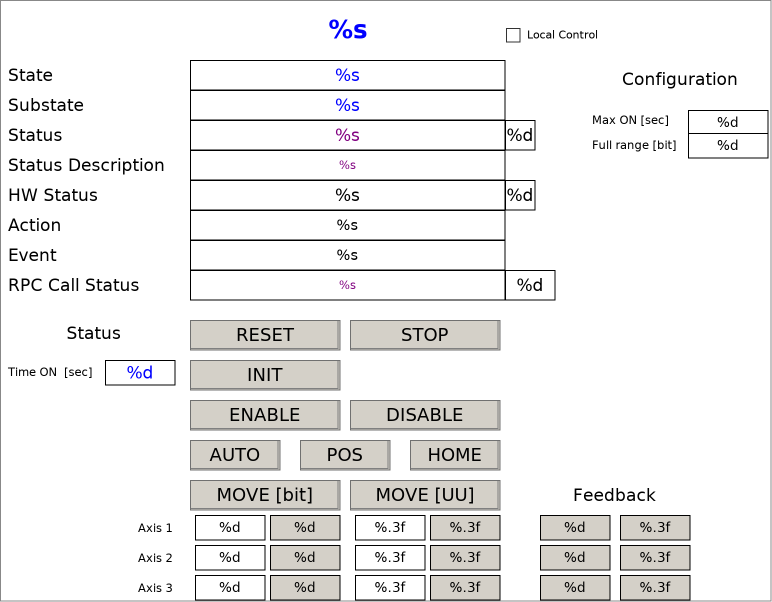
VISUALIZATION GUI_TEMPLATE_PIEZO  // 772x602
VAR_IN_OUT
	m_Instance:	FB_PIEZO_BASE;
END_VAR
    Rectangle (190,60 315x30), "%s", text variable: m_Instance.stat.sState
    Rectangle (190,90 315x30), "%s", text variable: m_Instance.stat.sSubstate
    Button (190,320 150x30), "RESET", input disabled if: (m_Instance.stat.bLocal = FALSE) <> 0
        OnMouseDown: execute { m_Instance.ctrl.nCommand := E_PIEZO_COMMAND.RESET; m_Instance.ctrl.bExecute := TRUE; }
    Button (190,360 150x30), "INIT", input disabled if: (m_Instance.stat.bLocal = FALSE) <> 0
        OnMouseDown: execute { m_Instance.ctrl.nCommand := E_PIEZO_COMMAND.INIT; m_Instance.ctrl.bExecute := TRUE; }
    Button (350,320 150x30), "STOP", input disabled if: (m_Instance.stat.bLocal = FALSE) <> 0
        OnMouseDown: execute { m_Instance.ctrl.nCommand := E_PIEZO_COMMAND.STOP; m_Instance.ctrl.bExecute := TRUE; }
    Button (190,400 150x30), "ENABLE", input disabled if: (m_Instance.stat.bLocal = FALSE) <> 0
        OnMouseDown: execute { m_Instance.ctrl.nCommand := E_PIEZO_COMMAND.ENABLE; m_Instance.ctrl.bExecute := TRUE; }
    Button (350,400 150x30), "DISABLE", input disabled if: (m_Instance.stat.bLocal = FALSE) <> 0
        OnMouseDown: execute { m_Instance.ctrl.nCommand := E_PIEZO_COMMAND.DISABLE; m_Instance.ctrl.bExecute := TRUE; }
    Button (190,440 90x30), "AUTO", tooltip "Start AUTO mode", input disabled if: (m_Instance.stat.bLocal = FALSE) <> 0
        OnMouseDown: execute { m_Instance.ctrl.nCommand := E_PIEZO_COMMAND.AUTO; m_Instance.ctrl.bExecute := TRUE; }
    Button (300,440 90x30), "POS", tooltip "Stop AUTO mode, if running. Keep piezos where they are.", input disabled if: (m_Instance.stat.bLocal = FALSE) <> 0
        OnMouseDown: execute { m_Instance.ctrl.nCommand := E_PIEZO_COMMAND.POS; m_Instance.ctrl.bExecute := TRUE; }
    Rectangle (5,60 180x30), "State"
    Rectangle (5,90 180x30), "Substate"
    Rectangle (190,120 315x30), "%s", text variable: m_Instance.stat.sStatus
    Rectangle (190,150 315x30), "%s", text variable: m_Instance.stat.sErrorText
    Rectangle (5,120 180x30), "Status"
    Rectangle (5,150 180x30), "Status Description"
    Rectangle (190,210 315x30), "%s", text variable: m_Instance.stat.sActionDesc
    Rectangle (190,240 315x30), "%s", text variable: m_Instance.stat.sEventDesc
    Rectangle (190,180 315x30), "%s", text variable: m_Instance.stat.sHwStatus
    Rectangle (5,180 180x30), "HW Status"
    Rectangle (505,180 30x30), "%d", tooltip "HW Status Index", text variable: m_Instance.stat.nHwStatus
    Rectangle (5,210 180x30), "Action"
    Rectangle (5,240 180x30), "Event"
    Rectangle (232,12 232x35), "%s", text variable: m_Instance.cfg.sName
    Rectangle (590,64 180x30), "Configuration"
    Rectangle (589,110 155x20), "Max ON [sec]"
    Rectangle (589,135 155x20), "Full range [bit]"
    Rectangle (688,110 80x25), "%d", tooltip "Maximum allowed time for lamp to be ON [sec] (>=0). Zero means no limit.", text variable: m_Instance.cfg.nMaxOn, input disabled if: (m_Instance.stat.bLocal = FALSE) <> 0
        OnMouseDown: write the text variable via Default, min 0
    Rectangle (688,133 80x25), "%d", tooltip "Full range of A/D converter controlling the intensity [bit]. Examples: 12 bit A/D = 4095 15 bit A/D = 32767 16 bit A/D = 65535", text variable: m_Instance.cfg.nFullRange[0].nValue, input disabled if: (m_Instance.stat.bLocal = FALSE) <> 0
        OnMouseDown: write the text variable via Default, min 0
    Checkbox (504,20 116x30), "Local Control", variable: m_Instance.stat.bLocal
    Rectangle (48,318 92x30), "Status"
    Rectangle (105,360 70x25), "%d", tooltip "Time since last ON command [sec]. Updated only if MaxON > 0.", text variable: m_Instance.stat.nTimeOn
    Rectangle (5,357 95x30), "Time ON [sec]"
    Rectangle (505,120 30x30), "%d", text variable: m_Instance.stat.nStatus
    Button (190,480 150x30), "MOVE [bit]", input disabled if: (m_Instance.stat.bLocal = FALSE) <> 0
        OnMouseDown: execute { m_Instance.ctrl.nCommand := E_PIEZO_COMMAND.MOVE_BIT; m_Instance.ctrl.bExecute := TRUE; }
    Rectangle (195,515 70x25), "%d", tooltip "Axis 1 Set Value [bit]", text variable: m_Instance.ctrl.nPosBit[0].nValue, input disabled if: (m_Instance.stat.bLocal = FALSE) <> 0
        OnMouseDown: write the text variable via Default
    Rectangle (195,545 70x25), "%d", tooltip "Axis 2 Set Value [bit]", text variable: m_Instance.ctrl.nPosBit[1].nValue, input disabled if: (m_Instance.stat.bLocal = FALSE) <> 0
        OnMouseDown: write the text variable via Default
    Button (350,480 150x30), "MOVE [UU]", input disabled if: (m_Instance.stat.bLocal = FALSE) <> 0
        OnMouseDown: execute { m_Instance.ctrl.nCommand := E_PIEZO_COMMAND.MOVE_USER; m_Instance.ctrl.bExecute := TRUE; }
    Rectangle (355,515 70x25), "%.3f", tooltip "Axis 1 Set position [UU]", text variable: m_Instance.ctrl.lrPosUser[0].lrValue, input disabled if: (m_Instance.stat.bLocal = FALSE) <> 0
        OnMouseDown: write the text variable via Default
    Rectangle (355,545 70x25), "%.3f", tooltip "Axis 2 Set position [UU]", text variable: m_Instance.ctrl.lrPosUser[1].lrValue, input disabled if: (m_Instance.stat.bLocal = FALSE) <> 0
        OnMouseDown: write the text variable via Default
    Rectangle (270,515 70x25), "%d", tooltip "Axis 1 Actual Output [bit]", text variable: m_Instance.q_nCtrl[0], input disabled if: TRUE
        OnMouseDown: write the text variable via Default, min 0
    Rectangle (270,545 70x25), "%d", tooltip "Axis 2 Actual Output [bit]", text variable: m_Instance.q_nCtrl[1], input disabled if: TRUE
        OnMouseDown: write the text variable via Default, min 0
    Rectangle (430,515 70x25), "%.3f", tooltip "Axis 1 Actual Output [UU]", text variable: m_Instance.stat.lrSetPosUsr[0].lrValue, input disabled if: TRUE
        OnMouseDown: write the text variable via Default, min 0
    Rectangle (430,545 70x25), "%.3f", tooltip "Axis 2 Actual Output [UU]", text variable: m_Instance.stat.lrSetPosUsr[1].lrValue, input disabled if: TRUE
        OnMouseDown: write the text variable via Default, min 0
    Button (410,440 90x30), "HOME", tooltip "Home piezos", input disabled if: (m_Instance.stat.bLocal = FALSE) <> 0
        OnMouseDown: execute { m_Instance.ctrl.nCommand := E_PIEZO_COMMAND.HOME; m_Instance.ctrl.bExecute := TRUE; }
    Rectangle (195,575 70x25), "%d", tooltip "Axis 3 Set Value [bit]", text variable: m_Instance.ctrl.nPosBit[2].nValue, input disabled if: (m_Instance.stat.bLocal = FALSE) <> 0
        OnMouseDown: write the text variable via Default
    Rectangle (355,575 70x25), "%.3f", tooltip "Axis 3 Set position [UU]", text variable: m_Instance.ctrl.lrPosUser[2].lrValue, input disabled if: (m_Instance.stat.bLocal = FALSE) <> 0
        OnMouseDown: write the text variable via Default
    Rectangle (270,575 70x25), "%d", tooltip "Axis 3 Actual Output [bit]", text variable: m_Instance.q_nCtrl[2], input disabled if: TRUE
        OnMouseDown: write the text variable via Default, min 0
    Rectangle (430,575 70x25), "%.3f", tooltip "Axis 3 Actual Output [UU]", text variable: m_Instance.stat.lrSetPosUsr[2].lrValue, input disabled if: TRUE
        OnMouseDown: write the text variable via Default, min 0
    Rectangle (135,518 55x20), "Axis 1"
    Rectangle (135,548 55x20), "Axis 2"
    Rectangle (135,578 55x20), "Axis 3"
    Rectangle (190,270 315x30), "%s", text variable: m_Instance.stat.sRpcErrorText
    Rectangle (5,270 180x30), "RPC Call Status"
    Rectangle (505,270 50x30), "%d", tooltip "RPC Error Code 0 - OK", text variable: m_Instance.stat.nRpcErrorCode
    Rectangle (540,515 70x25), "%d", tooltip "Axis 1 Feedback [bit]", text variable: m_Instance.stat.nActPosBit[0].nValue, input disabled if: TRUE
        OnMouseDown: write the text variable via Default, min 0
    Rectangle (550,480 129x30), "Feedback"
    Rectangle (620,515 70x25), "%.3f", tooltip "Axis 1 Feedback [UU]", text variable: m_Instance.stat.lrActPosUsr[0].lrValue, input disabled if: TRUE
        OnMouseDown: write the text variable via Default, min 0
    Rectangle (540,545 70x25), "%d", tooltip "Axis 2 Feedback [bit]", text variable: m_Instance.stat.nActPosBit[1].nValue, input disabled if: TRUE
        OnMouseDown: write the text variable via Default, min 0
    Rectangle (620,545 70x25), "%.3f", tooltip "Axis 2 Feedback [UU]", text variable: m_Instance.stat.lrActPosUsr[1].lrValue, input disabled if: TRUE
        OnMouseDown: write the text variable via Default, min 0
    Rectangle (540,575 70x25), "%d", tooltip "Axis 3 Feedback [bit]", text variable: m_Instance.stat.nActPosBit[2].nValue, input disabled if: TRUE
        OnMouseDown: write the text variable via Default, min 0
    Rectangle (620,575 70x25), "%.3f", tooltip "Axis 3 Feedback [UU]", text variable: m_Instance.stat.lrActPosUsr[2].lrValue, input disabled if: TRUE
        OnMouseDown: write the text variable via Default, min 0
END_VISUALIZATION

(* stored: Version 1.1.0.1, ProductVersion 3.1.4022.16
   Visu GUI_TEMPLATE_PIEZO: Id {208abcb1-f1a3-4a00-92a5-f362cd7556ac} *)
